FUNCTION_BLOCK FB_ModbusMaster

VAR
	MB: ModbusRtuMaster_KL6x22B;
	
	nReadRegsVals: POINTER TO ARRAY[1..10] OF WORD;
	nWriteRegVals: ARRAY[1..10] OF WORD;
	
	
	bRequestFinshed : POINTER TO BOOL;
		
	nSlaveAddress : BYTE;
	nQtyWordsToRead : WORD;
	nQtyWordsToWrite : WORD;
	nAdrFirstSlaveRegisterRead : WORD;
	nAdrFirstSlaveRegisterWrite : WORD;
	nTimeout : TIME := T#5S;
	
	
	// State Machine
	eState: (IDLE, BUSY, ERROR) := IDLE;
	eSMtate: (WAIT, READ_TRIG, READ, WRITE_TRIG, WRITE, ERROR) := WAIT;
	eSMState_prev:  (WAIT, READ_TRIG, READ, WRITE_TRIG, WRITE, ERROR) := WAIT;
	bBusy: BOOL;
	
	//eOperationType: (READ_OP, WRITE_OP, READWRITE_OP);
	eOperationType: E_AccessType;
	fbTrigger : R_TRIG;
	
	bOperationFirstRun: BOOL := TRUE;
	nNumRetries: INT := 0; 
	nRetryThreshold: INT := 10;

END_VAR

fbTrigger();

CASE eState OF
	WAIT :
		eState := IDLE;
		MB.ReadRegs(Execute := FALSE);
        MB.WriteRegs(Execute := FALSE);
	
		
		IF fbTrigger.Q THEN
			IF eOperationType = E_AccessType.WRITE THEN
				eSMtate := WRITE_TRIG;
			ELSIF eOperationType = E_AccessType.READ THEN
				eSMtate := READ_TRIG;
			END_IF
		END_IF
		
		
		
	READ_TRIG : 
		eState := BUSY;
		IF bOperationFirstRun THEN
			nNumRetries := 0;
			bOperationFirstRun := FALSE;
		END_IF
	
		IF eOperationType = E_AccessType.READ THEN
			
			 MB.ReadRegs(
				UnitID:= nSlaveAddress, 
				Quantity:= nQtyWordsToRead, 
				MBAddr:= nAdrFirstSlaveRegisterRead, 
				cbLength:= nQtyWordsToRead * 2,//SIZEOF(nReadRegsVals), 
				pMemoryAddr:= ADR(nReadRegsVals), 
				Execute:= TRUE, 
				Timeout:= nTimeout );
			
			
			IF NOT MB.BUSY THEN 
				MB.ReadRegs(Execute := FALSE );
				bBusy := TRUE;
				IF MB.Error THEN 
					eSMState_prev := eSMtate;
					eSMtate := ERROR;           // handle errors 
				ELSE 
					eSMtate := READ; // [...]               // keep going 
				END_IF
			END_IF
		END_IF
		
		
	READ :
	
		IF NOT MB.BUSY THEN
			eSMtate := WAIT;
			bRequestFinshed^ := TRUE;
			bBusy := FALSE;
			fbTrigger.CLK := FALSE;
			bOperationFirstRun := TRUE;
		ELSIF MB.Error THEN
			eSMState_prev := eSMtate;
			eSMtate := ERROR;
		END_IF
	
	
	
	WRITE_TRIG :

		IF bOperationFirstRun THEN
			nNumRetries := 0;
			bOperationFirstRun := FALSE;
		END_IF
	(*
		MB.WriteRegs(
			UnitID:= nSlaveAddress, 
			Quantity:= nQtyWordsToWrite, 
			MBAddr:= nAdrFirstSlaveRegisterWrite, 
			cbLength:= nQtyWordsToWrite * 2, 
			pMemoryAddr:= ADR(nWriteRegVals), 
			Execute:= TRUE, 
			Timeout:= nTimeout); 
		*)	
		
		MB.UnitID:= nSlaveAddress;
		MB.Quantity:=1;
		MB.MBAddr:= nAdrFirstSlaveRegisterWrite;
		MB.cbLength:= nQtyWordsToWrite * 2;
		MB.pMemoryAddr:= ADR(nWriteRegVals);
		MB.Execute:= TRUE;
		MB.Timeout:= nTimeout;
		MB.WriteSingleRegister();
		
			
		IF NOT MB.BUSY THEN 
			//MB.WriteRegs(Execute := FALSE );
			MB.Execute := FALSE;
			bBusy := TRUE;
			IF MB.Error THEN 
				eSMState_prev := eSMtate;
				eSMtate := ERROR;           				// handle errors 
			ELSE 
				eSMtate := WRITE;			            // keep going 
			END_IF
		END_IF

	
		
	WRITE:
		IF NOT MB.BUSY THEN
			eSMtate := WAIT;
			bRequestFinshed^ := TRUE;
			bBusy := FALSE;
			fbTrigger.CLK := FALSE;
			bOperationFirstRun := TRUE;
		ELSIF MB.Error THEN
			eSMState_prev := eSMtate;
			eSMtate := ERROR;
		END_IF
	
		
	ERROR:
		nNumRetries := nNumRetries + 1;
		IF nNumRetries > nRetryThreshold THEN
			eState := ERROR;
		ELSE
			eSMtate := eSMState_prev;
		END_IF
		 
			
		

END_CASE

METHOD Error : BOOL
VAR_INPUT
END_VAR
Error := MB.Error;
END_METHOD

METHOD FB_init : BOOL
VAR_INPUT
	bInitRetains : BOOL; // if TRUE, the retain variables are initialized (warm start / cold start)
	bInCopyCode : BOOL;  // if TRUE, the instance afterwards gets moved into the copy code (online change)
END_VAR
END_METHOD

METHOD isBusy : BOOL
isBusy := bBusy;
END_METHOD

METHOD readRegs : BOOL
VAR_INPUT
	
	ReadRegsVals: POINTER TO ARRAY[1..10] OF WORD;
	SlaveAddress : UINT;
	QtyWordsToRead : UINT;
	AdrFirstSlaveRegisterRead : UINT;
	bRequestCompleted : POINTER TO BOOL;
	
END_VAR

VAR_OUTPUT
	bRequestAccepted: BOOL;
END_VAR
IF eState = WAIT THEN
	eOperationType := E_AccessType.READ;
	nReadRegsVals := ReadRegsVals;
	nSlaveAddress := UINT_TO_BYTE(SlaveAddress);
	nQtyWordsToRead := UINT_TO_WORD(QtyWordsToRead);
	nAdrFirstSlaveRegisterRead := UINT_TO_WORD(AdrFirstSlaveRegisterRead);
	fbTrigger.CLK := TRUE;
	bRequestAccepted := TRUE;
	bBusy := TRUE;
	bRequestFinshed := bRequestCompleted;
END_IF
END_METHOD

METHOD writeReg : BOOL
VAR_INPUT
	WriteRegVal: WORD;
	SlaveAddress : UINT;
	AdrFirstSlaveRegisterWrite : UINT;
	bRequestCompleted : POINTER TO BOOL;
END_VAR

VAR_OUTPUT
	bRequestAccepted: BOOL := FALSE;
END_VAR

IF eState = WAIT THEN
	eOperationType := E_AccessType.WRITE;
	nWriteRegVals[1] := WriteRegVal;
	nSlaveAddress := UINT_TO_BYTE(SlaveAddress);
	nQtyWordsToWrite := 1;
	nAdrFirstSlaveRegisterWrite := UINT_TO_BYTE(AdrFirstSlaveRegisterWrite);
	bRequestAccepted := TRUE;
	bRequestFinshed := bRequestCompleted;
	fbTrigger.CLK := TRUE;
	eState := WRITE_TRIG;
	
END_IF
END_METHOD

METHOD writeRegs : BOOL
VAR_INPUT

	WriteRegVals: ARRAY[1..10] OF WORD;
	
	SlaveAddress : UINT;
	QtyWordsToWrite : UINT;
	AdrFirstSlaveRegisterWrite : UINT;
	bRequestCompleted: POINTER TO BOOL;

END_VAR

VAR_OUTPUT
	bRequestAccepted: BOOL := FALSE;
END_VAR
IF eState = WAIT THEN
	eOperationType := E_AccessType.WRITE;
	nWriteRegVals := WriteRegVals;
	nSlaveAddress := UINT_TO_BYTE(SlaveAddress);
	nQtyWordsToWrite := UINT_TO_WORD(QtyWordsToWrite);
	nAdrFirstSlaveRegisterWrite := UINT_TO_WORD(AdrFirstSlaveRegisterWrite);
	fbTrigger.CLK := TRUE;
	bRequestAccepted := TRUE;
	bRequestFinshed := bRequestCompleted;
	eState := WRITE_TRIG;
END_IF
END_METHOD

END_FUNCTION_BLOCK

(* stored: Version 1.1.0.1, ProductVersion 3.1.4024.12
   POU FB_ModbusMaster: Id {e0b53259-e081-4754-a027-d87bf9b01c91}, SpecialFunc None
   Method Error: Id {1ba917d6-d711-4350-a108-0591f997f8a1}
   Method FB_init: Id {1d28eff9-e697-4725-9f04-e098dd7679cc}
   Method isBusy: Id {723204d6-2503-44fb-bd27-abfca00f7695}
   Method readRegs: Id {86acfe3a-6c2c-4699-b47b-d6f78a629193}
   Method writeReg: Id {72eaa5db-9247-4fc8-8f50-59c4535b231c}
   Method writeRegs: Id {9913fe0a-499f-4d82-b327-421f60fe5e77} *)
